{attribute 'qualified_only'}
TYPE E_MemCmpResults :
(
	pBUFF1_LESS_THAN_pBUFF2	:= -1,
	IDENTICAL	:= 0,
	PbUFF1_GREATER_THAN_pBUFF2	:= 1,
	ERROR	:= 255
)DINT;
END_TYPE

(* stored: Version 1.1.0.1, ProductVersion 3.1.4024.13
   DUT E_MemCmpResults: Id {2dcaf930-168a-0ef9-2ea9-9722efba1aff} *)
